TYPE JobData :
STRUCT
	gridPointGoal : GridPoint;
	goalRotation : LREAL;
	goalGripper : GripperCmd;
END_STRUCT
END_TYPE

(* stored: Version 1.1.0.1, ProductVersion 3.1.4024.11
   DUT JobData: Id {4922dc58-7aaa-459b-9984-d44dabc77b2c} *)
